{attribute 'linkalways'} 
{attribute 'no_explicit_call' := 'This FB is a CLASS and must be accessed using methods or properties'}
{attribute 'enable_dynamic_creation'}
FUNCTION_BLOCK _ETcVnConnectedComponentsAlgorithm EXTENDS EnumDatatypeBase
VAR
	localData : ETcVnConnectedComponentsAlgorithm;
	activeData : REFERENCE TO ETcVnConnectedComponentsAlgorithm;
	enumBaseDatatype : _DINT(localData);
END_VAR

METHOD PRIVATE AddLocalEnumeration
VAR_INPUT
	Enumeration : T_MAXSTRING;
	Value : ETcVnConnectedComponentsAlgorithm;
END_VAR
AddEnumeration(Enumeration, Value);
END_METHOD

PROPERTY PUBLIC Address : PVOID
GET
Address := ADR(activeData);
END_GET
END_PROPERTY

METHOD PUBLIC ClearReference
VAR_INPUT
END_VAR
activeData REF= localData;
SetBaseDatatypeReference();
END_METHOD

METHOD PUBLIC Clone : I_Datatype
VAR
    pClone : POINTER TO _ETcVnConnectedComponentsAlgorithm;
END_VAR
pClone := __NEW(_ETcVnConnectedComponentsAlgorithm(InitialValue := Value));
Clone := pClone^;
END_METHOD

METHOD FB_init : BOOL
VAR_INPUT
	bInitRetains : BOOL; // if TRUE, the retain variables are initialized (warm start / cold start)
	bInCopyCode : BOOL;  // if TRUE, the instance afterwards gets moved into the copy code (online change)
	InitialValue : ETcVnConnectedComponentsAlgorithm;
END_VAR
localData := InitialValue;
AddBaseDatatype(enumBaseDatatype);
ClearReference();

AddLocalEnumeration('TCVN_CCA_WU', ETcVnConnectedComponentsAlgorithm.TCVN_CCA_WU);
AddLocalEnumeration('TCVN_CCA_GRANA', ETcVnConnectedComponentsAlgorithm.TCVN_CCA_GRANA);
END_METHOD

PROPERTY PUBLIC Identifier : T_MAXSTRING
GET
Identifier := 'ETcVnConnectedComponentsAlgorithm';
END_GET
END_PROPERTY

METHOD IsEnumeratorValueEqual : BOOL
VAR_INPUT
	Enumerator : I_KeyValueForwardEnumerator;
END_VAR
VAR
	storedValue : ETcVnConnectedComponentsAlgorithm;
END_VAR
IF NOT Enumerator.TryGet(storedValue) THEN
	RETURN;
END_IF

IsEnumeratorValueEqual := storedValue = activeData;
END_METHOD

METHOD PUBLIC MakeReferenceTo
VAR_INPUT
	ReferenceTarget : REFERENCE TO ETcVnConnectedComponentsAlgorithm;
END_VAR
activeData REF= ReferenceTarget;
SetBaseDatatypeReference();
END_METHOD

METHOD PROTECTED SetBaseDatatypeReference
VAR_INPUT
END_VAR
enumBaseDatatype.MakeReferenceTo(activeData);
END_METHOD

PROPERTY PUBLIC Size : UDINT
GET
Size := SIZEOF(activeData);
END_GET
END_PROPERTY

METHOD TryMakeReferenceTo : BOOL
VAR_INPUT
	Target : I_Datatype;
END_VAR
VAR
	targetAsEnum : I_EnumDatatype;
	pTargetData : POINTER TO ETcVnConnectedComponentsAlgorithm;
END_VAR
IF NOT Target.TryResolveAsEnumDatatype(targetAsEnum) THEN
	RETURN;
END_IF

IF targetAsEnum.Identifier <> Identifier THEN
	RETURN;
END_IF

pTargetData := Target.Address;
activeData REF= pTargetData^;
SetBaseDatatypeReference();
TryMakeReferenceTo := TRUE;
END_METHOD

PROPERTY PUBLIC Value : ETcVnConnectedComponentsAlgorithm
GET
Value := activeData;
END_GET
SET
activeData := Value;
END_SET
END_PROPERTY

END_FUNCTION_BLOCK

(* stored: Version 1.1.0.1, ProductVersion 3.1.4024.12
   POU _ETcVnConnectedComponentsAlgorithm: Id {0ebbb17c-5356-4b43-a669-66bf4a23c0ec}, SpecialFunc None
   Folder Constructor: Id {d269f08d-cda1-4bf8-84a9-94d85504a34b}
   Folder Private: Id {0a3efd4d-41da-454d-a51c-9e8e151682ac}
   Folder Protected: Id {1cf1f4be-7007-4cab-9c7a-93d51d01701d}
   Method AddLocalEnumeration: Id {8f643058-27f8-4ca7-90aa-30570f51bf6f}
   Property Address: Id {b6441540-b0b3-40bc-9d21-97639b1a4560}
   Get Get: Id {c4736b23-2b6c-4a1f-91c3-7318079ca9f8}
   Method ClearReference: Id {e6919e26-dc71-43b9-a5e0-9bed6097153a}
   Method Clone: Id {b9f60cc9-a283-4084-95e1-24086af86e29}
   Method FB_init: Id {20659b03-bbd7-4110-9a70-452bfc830a8b}
   Property Identifier: Id {705a9f5f-cce4-4534-8035-aea1c75e42b0}
   Get Get: Id {9d8bfea7-704e-4fb4-99be-7f3cc5627159}
   Method IsEnumeratorValueEqual: Id {7c97b15a-1d78-465b-b134-ba120645da42}
   Method MakeReferenceTo: Id {af004e7f-62eb-415f-b159-713e7bbf90b4}
   Method SetBaseDatatypeReference: Id {d91f07cd-39b7-45b4-a1b8-2e25ff2a1d9e}
   Property Size: Id {48a9009a-4048-43c3-aeac-7c0f2142f116}
   Get Get: Id {d49abea5-64b1-47e5-bf65-0a7ccf392537}
   Method TryMakeReferenceTo: Id {b877e867-7b51-4577-8b4b-2d87c00de3cd}
   Property Value: Id {93b8b3de-b0e0-49f9-80cc-b1e14b92447e}
   Get Get: Id {9e46b26f-6d42-463f-8211-5d2bb28a9462}
   Set Set: Id {70c8dfcb-5090-4da0-8524-d3a59a9119ce} *)
